FUNCTION_BLOCK ABSTRACT FB_AbstractObserver EXTENDS FB_Object IMPLEMENTS I_Observer
VAR
    _nTypeClass:        __SYSTEM.TYPE_CLASS;
    _pVal:              POINTER TO BYTE;
    _nSize:             DINT;
    _nUpdateCounter:    UDINT;
END_VAR

METHOD PROTECTED _Update
VAR_INPUT
    pData:          POINTER TO BYTE;
    nTypeClass:     __SYSTEM.TYPE_CLASS;
    nSize:          UDINT;
END_VAR
VAR
    nMemcpyRes:     UDINT;
END_VAR
IF nTypeClass <> THIS^._nTypeClass THEN
    RETURN;
END_IF

IF nSize <> TO_UDINT(THIS^._nSize) THEN
    RETURN;
END_IF

IF pData = 0 THEN
    RETURN;
END_IF

nMemcpyRes := Tc2_System.MEMCPY(destAddr := THIS^._pVal,
                                srcAddr := pData,
                                n := TO_UDINT(THIS^._nSize));

IF nMemcpyRes <> 0 THEN
    THIS^._nUpdateCounter := THIS^._nUpdateCounter + 1;
END_IF
END_METHOD

PROPERTY nTypeClass : __SYSTEM.TYPE_CLASS
GET
nTypeClass := THIS^._nTypeClass;
END_GET
END_PROPERTY

METHOD PROTECTED PostUpdate
VAR_INPUT
END_VAR
END_METHOD

METHOD PROTECTED PreUpdate
VAR_INPUT
END_VAR
END_METHOD

{attribute 'hasanytype'}
METHOD FINAL Update
(* Template method for updating using ANY-typed variable *)
VAR_INPUT
    anyVal:         ANY;
END_VAR
THIS^.PreUpdate();

THIS^._Update(pData := anyVal.pValue,
              nTypeClass := anyVal.TypeClass,
              nSize := TO_UDINT(anyVal.diSize));

THIS^.PostUpdate();
END_METHOD

METHOD FINAL UpdateP
(* Template method for updating using explicit
   variable information *)
VAR_INPUT
    pData:          POINTER TO BYTE;
    nTypeClass:     __SYSTEM.TYPE_CLASS;
    nSize:          UDINT;
END_VAR
THIS^.PreUpdate();

THIS^._Update(pData := pData,
              nTypeClass := nTypeClass,
              nSize := nSize);

THIS^.PostUpdate();
END_METHOD

END_FUNCTION_BLOCK

(* stored: Version 1.1.0.1, ProductVersion 3.1.4024.12
   POU FB_AbstractObserver: Id {59366400-b2f5-4598-9c5c-2530302a1d7f}, SpecialFunc None
   Method _Update: Id {04601ce4-ef10-086c-2ba8-698f7bbc7727}
   Property nTypeClass: Id {fde940e3-79f9-098e-0135-d3adf4a5926d}
   Get Get: Id {8c43525e-7ffb-0f69-01a8-b6b495032969}
   Method PostUpdate: Id {30236f96-dbe0-0ab4-0064-2829402f1028}
   Method PreUpdate: Id {dc87cb06-4c62-0279-1d2a-b00e97977a5f}
   Method Update: Id {db1aebf2-fca2-494e-a52a-f9c476d5cd33}
   Method UpdateP: Id {754e5201-247b-4bda-8c15-e31312212f2e} *)
